FUNCTION_BLOCK SUB_SINT (* IEC 61131-3 SINT Subtraction *)
  (* Standard: 61131-3 *)
  (* Version 0.0, 2004-12-15, JHC, Rockwell Automation, Converted from SRC format. *)
  (* Compiler header: package fb.rt.plc.math; *)
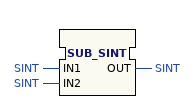
  VAR_INPUT
    IN1 : SINT; (* Minuend *)
    IN2 : SINT; (* Subtrahend *)
  END_VAR
  VAR_OUTPUT
    OUT : SINT; (* Difference *)
  END_VAR
END_FUNCTION_BLOCK
